{attribute 'OPC.UA.DA.StructuredType' := '1'}
	{attribute 'OPC.UA.DA' := '1'}
TYPE ST_EyesSpecific :
STRUCT
    Result          : STRING(255) := '';

END_STRUCT
END_TYPE

(* stored: Version 1.1.0.1, ProductVersion 3.1.4026.18
   DUT ST_EyesSpecific: Id {ccd32ea7-61fc-43f3-adf5-9241d9e87f01} *)
